// Implicitly generated code : DO NOT EDIT
FUNCTION CheckDivLInt : LINT
VAR_INPUT
    divisor:LINT;
END_VAR


// Implicitly generated code : Only an Implementation suggestion
{noflow}
IF divisor = 0 THEN
    CheckDivLInt:=1;
ELSE
    CheckDivLInt:=divisor;
END_IF;
{flow}

END_FUNCTION

(* stored: Version 1.1.0.1
   POU CheckDivLInt: Id {2a9a0768-801b-4379-9602-cc3f9bfe0176}, SpecialFunc CheckDivInt64 *)
